(* CODESYS project OPC UA on Raspberry Pi.project

Project tree, tasks and I/O mapping:
  Device : CODESYS Control for Raspberry Pi, 3S - Smart Software Solutions GmbH, version 3.5.11.20
    application Application
      libraries: Standard, * (System)
      task MainTask (cyclic, interval 4 ms, priority 1) calls PLC_PRG
      program PLC_PRG [CFC]
      Symbols
    SoftMotion General Axis Pool
    I²C
    SPI
    GPIOs_A_B : GPIOs A/B, 3S - Smart Software Solutions GmbH, version 3.5.11.0
        unmapped channels: digital inputs (GPIO0..GPIO31), digital outputs (GPIO0..GPIO31)
    Onewire
    Camera device
      <Leer>
*)

// Device/Application/PLC_PRG
PROGRAM PLC_PRG
VAR
	piface_eingang_1: BOOL;
	piface_eingang_2: BOOL;
	piface_ausgang_1: BOOL;
END_VAR

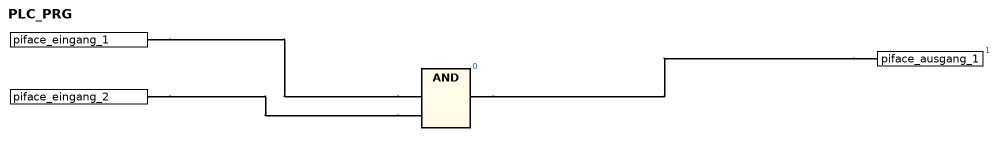
piface_ausgang_1 := piface_eingang_1 AND piface_eingang_2;

END_PROGRAM
